PROGRAM Stn055_61_Stn611MainMergePrestop
VAR
	
	{attribute 'TcLinkToOSO' := '.iPuckPresent   :=  <0,1,2>TIIB[N12S00 (AL1332)]^N12S03 (AL2341)^TxPDO^input byte 0;
								 .iBufferFull  :=  <0,1,2>TIIB[N12S00 (AL1332)]^N12S03 (AL2341)^TxPDO^input byte 2;
								 .oStopLower   :=  <0,1,1>TIIB[N12S00 (AL1332)]^N12S02 (EX260)^RxPDO^output byte 1'}
	fbConvStop: FB_ConvStop;
	
END_VAR

//  This code instantiates a component that is implimented as a common function block
//    Note that I/O is linked directly to I/O variables inside the named instance

gStn055_61_Stn611MainMergePrestop.ConvRunning := gConsumed_SafetyInterfaceConv.MtrRunning.Enc051Mtr05;

fbConvStop(
	pStn := ADR(gStn055),
	pCmp := ADR(gStn055_61_Stn611MainMergePrestop),
	pUpstreamStop := 0,
	pStateTraceBuffer := ADR(gStn055_StateTraceBuffer),
	pStateTraceFifo := ADR(gStn055_StateTraceFifo),
	pStats := ADR(gStn055_02_Stats));

END_PROGRAM

(* stored: Version 1.1.0.1, ProductVersion 3.1.4024.6
   POU Stn055_61_Stn611MainMergePrestop: Id {f0ae5a9f-ed8a-42af-8e57-e21d35be7306}, SpecialFunc None *)
